TYPE ST_ProductHandlingMachPar :
STRUCT
	GantryA						: ST_GantryMachPar;
	GantryB						: ST_GantryMachPar;
	CommisioningMode 			: BOOL	:= FALSE;
END_STRUCT
END_TYPE

(* stored: Version 1.1.0.1, ProductVersion 3.1.4020.12
   DUT ST_ProductHandlingMachPar: Id {948cd65e-9bb0-4941-be00-ae54532153c6} *)
